FUNCTION_BLOCK FB_LoadingStationA
VAR_INPUT
END_VAR
VAR_OUTPUT
END_VAR
VAR
END_VAR

END_FUNCTION_BLOCK

(* stored: Version 1.1.0.1
   POU FB_LoadingStationA: Id {19675339-fb1f-4115-a918-4decd2ed905a}, SpecialFunc None *)
